FUNCTION_BLOCK FB_Cinta_SFC  EXTENDS FB_Controller_SFC
VAR_INPUT
	IC: BOOL;
	Execute: BOOL;
	Ack: BOOL;
END_VAR
VAR_OUTPUT
	Ready: BOOL;
	Failure: BOOL;
	Done: BOOL;
END_VAR
VAR
END_VAR

VAR_INPUT
	RUN: BOOL;
	REV: BOOL;
	pp: BOOL;
	situar: BOOL;
	transportar: BOOL;
END_VAR
VAR_OUTPUT
END_VAR
VAR

END_VAR

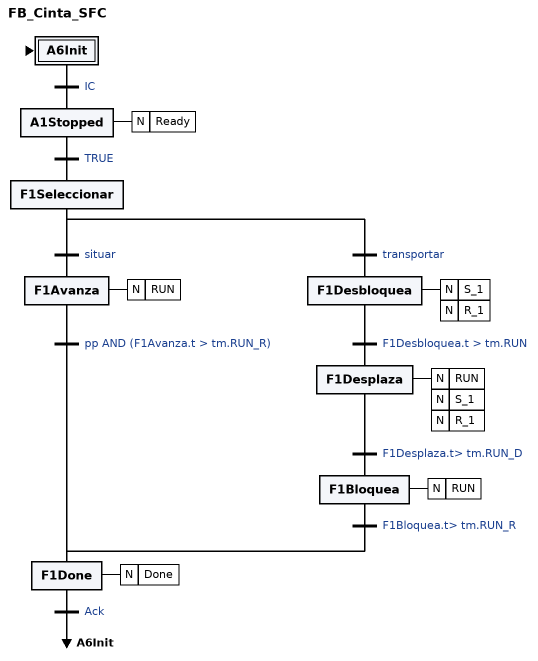
INITIAL_STEP A6Init:
END_STEP
TRANSITION FROM A6Init TO A1Stopped
    := IC;
END_TRANSITION
STEP A1Stopped:
    Ready(N);
END_STEP
TRANSITION FROM A1Stopped TO F1Seleccionar
    := TRUE;
END_TRANSITION
STEP F1Seleccionar:
END_STEP
TRANSITION FROM F1Seleccionar TO F1Avanza
    := situar;
END_TRANSITION
STEP F1Avanza:
    RUN(N);
END_STEP
TRANSITION FROM F1Avanza TO F1Done
    := pp AND (F1Avanza.t > tm.RUN_R);
END_TRANSITION
TRANSITION FROM F1Seleccionar TO F1Desbloquea
    := transportar;
END_TRANSITION
STEP F1Desbloquea:
    S_1(N);
    R_1(N);
END_STEP
TRANSITION FROM F1Desbloquea TO F1Desplaza
    := F1Desbloquea.t > tm.RUN;
END_TRANSITION
STEP F1Desplaza:
    RUN(N);
    S_1(N);
    R_1(N);
END_STEP
TRANSITION FROM F1Desplaza TO F1Bloquea
    := F1Desplaza.t> tm.RUN_D;
END_TRANSITION
STEP F1Bloquea:
    RUN(N);
END_STEP
TRANSITION FROM F1Bloquea TO F1Done
    := F1Bloquea.t> tm.RUN_R;
END_TRANSITION
STEP F1Done:
    Done(N);
END_STEP
TRANSITION FROM F1Done TO A6Init
    := Ack;
END_TRANSITION

END_FUNCTION_BLOCK

(* stored: Version 1.1.0.1, ProductVersion 3.1.4024.6
   POU FB_Cinta_SFC: Id {7a4e0e2e-bc1d-4eb2-80cf-952f4dd5e6da}, SpecialFunc None *)
